// TwinCAT 3 PLC project ph_lv0
// Title: tclib_ph_lv0
// Company: Poh
// Author: Poh
// ProjectVersion: 0.1.2.0
// ProgramVersion: 3.1.4020.1
// project tree:
//   Lv0_Components/Class/ C_STREAM.TcPOU, E_SEEK_STYLE.TcDUT
//   Lv0_Components/Data Definitions/Generic Return Code/ RETURN_CODE.TcDUT, LV0_RETURNCODE.TcGVL
//   Lv0_Components/Modules/ M_TRIGGERS.TcPOU
//   Version/ Global_Version.TcGVL
// real-time tasks:
//   TASK PlcTask: cycle T#10ms, priority 20, ADS port 350
//   TASK Fast: cycle T#3ms, priority 1, ADS port 351

// ---- Lv0_Components/Class/E_SEEK_STYLE.TcDUT
{attribute 'qualified_only'}
{attribute 'strict'}
TYPE E_SEEK_STYLE :
(
	E_STREAM_BEGIN := 0,
	E_STREAM_CURRENT,
	E_STREAM_END
);
END_TYPE

// ---- Lv0_Components/Data Definitions/Generic Return Code/RETURN_CODE.TcDUT
TYPE RETURN_CODE : DINT; END_TYPE

// ---- Lv0_Components/Data Definitions/Generic Return Code/LV0_RETURNCODE.TcGVL
(*
	Y:2016	M:0005	D:0011
	Library conventions:
	Values less than 0 represent success/success code 
	Values equal to 0 represent a busy return code
	Values more than 0 represent error/error codes 
*)
{attribute 'qualified_only'}
VAR_GLOBAL CONSTANT
	RETURN_SUCCESS 	: RETURN_CODE := -1;
	RETURN_BUSY		: RETURN_CODE := 0;
	RETURN_ERROR	: RETURN_CODE := 1;
END_VAR

// ---- Version/Global_Version.TcGVL
{attribute 'TcGenerated'}
// This function has been automatically generated from the project information.
VAR_GLOBAL CONSTANT
	{attribute 'const_non_replaced'}
	{attribute 'linkalways'}
	stLibVersion_tclib_ph_lv0 : ST_LibVersion := (iMajor := 0, iMinor := 1, iBuild := 2, iRevision := 0, sVersion := '0.1.2.0');
END_VAR

// ---- Lv0_Components/Class/C_STREAM.TcPOU
FUNCTION_BLOCK C_STREAM
VAR_INPUT
END_VAR
VAR_OUTPUT
END_VAR
VAR
	_StreamSize 			: UDINT;
	_StreamData 			: POINTER TO BYTE;
	_StreamPointingPosition	: UDINT;
END_VAR

PROPERTY Base_Data : POINTER TO BYTE
GET
Base_Data := _StreamData;
END_GET
SET
_StreamData := Base_Data;
END_SET
END_PROPERTY

METHOD Clear : RETURN_CODE
VAR_INPUT
END_VAR
VAR
	_i : UDINT;
END_VAR
FOR _i := 0 TO THIS^._StreamSize - 1 BY 1 DO
	THIS^._StreamData[_i] := 0;
END_FOR
_StreamPointingPosition := 0;
_StreamFilledPosition := 0;
Clear := LV0_RETURNCODE.RETURN_SUCCESS;
END_METHOD

METHOD FB_init : BOOL
VAR_INPUT
	bInitRetains : BOOL; // if TRUE, the retain variables are initialized (warm start / cold start)
	bInCopyCode : BOOL;  // if TRUE, the instance afterwards gets moved into the copy code (online change)
	Base_Stream : POINTER TO BYTE;
	Base_StreamSize : UDINT;
END_VAR
THIS^._StreamData := Base_Stream;
THIS^._StreamSize := Base_StreamSize;
END_METHOD

METHOD Peek : Byte
VAR_INPUT
END_VAR
Peek := _StreamData[_StreamPointingPosition];
END_METHOD

PROPERTY Position : UDINT
GET
Position := _StreamPointingPosition;
END_GET
END_PROPERTY

METHOD Read : RETURN_CODE
VAR_INPUT
	OUT_DATA : POINTER TO BYTE;
	OUT_SIZE : UDINT;
END_VAR
VAR 
	_i : UDINT;
END_VAR
IF _StreamPointingPosition + OUT_SIZE > _StreamSize - 1 THEN
	Read := LV0_RETURNCODE.RETURN_ERROR;
	RETURN;
END_IF

FOR _i := 0 TO OUT_SIZE - 1 BY 1 DO
	OUT_DATA[_i] := _StreamData[_StreamPointingPosition];
	_StreamPointingPosition := _StreamPointingPosition + 1;
END_FOR
END_METHOD

METHOD Seek : RETURN_CODE
VAR_INPUT
	Offset 		: UDINT;
	SeekMode 	: E_SEEK_STYLE;
END_VAR
CASE SeekMode OF
E_SEEK_STYLE.E_STREAM_BEGIN:
	IF Offset > _StreamSize - 1 THEN
		Seek := 1 * LV0_RETURNCODE.RETURN_ERROR;
		RETURN;
	END_IF
	_StreamPointingPosition := Offset;
E_SEEK_STYLE.E_STREAM_CURRENT:
	IF _StreamPointingPosition + Offset > _StreamSize - 1 THEN
		Seek := 2 * LV0_RETURNCODE.RETURN_ERROR;
		RETURN;
	END_IF
	_StreamPointingPosition := _StreamPointingPosition + Offset;
E_SEEK_STYLE.E_STREAM_END:
	IF Offset > _StreamSize - 1 THEN
		Seek := 3 * LV0_RETURNCODE.RETURN_ERROR;
		RETURN;
	END_IF
	_StreamPointingPosition := _StreamSize - 1 - Offset;
END_CASE

Seek := LV0_RETURNCODE.RETURN_SUCCESS;
RETURN;
END_METHOD

PROPERTY Stream_Size : UDINT
GET
Stream_Size := _StreamSize;
END_GET
SET
_StreamSize := Stream_Size;
END_SET
END_PROPERTY

METHOD Write : RETURN_CODE
VAR_INPUT
	IN_DATA : POINTER TO BYTE;
	IN_SIZE : UDINT;
END_VAR
VAR 
	_i : UDINT;
END_VAR
IF _StreamPointingPosition + IN_SIZE > _StreamSize - 1 THEN
	//Buffer size insufficient.
		Write := LV0_RETURNCODE.RETURN_ERROR;
		RETURN;
END_IF

FOR _i := 0 TO IN_SIZE - 1 BY 1 DO
	_StreamData[_StreamPointingPosition] := IN_DATA[_i];
	_StreamPointingPosition := _StreamPointingPosition + 1;
END_FOR

Write := LV0_RETURNCODE.RETURN_SUCCESS;
RETURN;
END_METHOD

END_FUNCTION_BLOCK

// ---- Lv0_Components/Modules/M_TRIGGERS.TcPOU
(*
	Y:2016		M:05		D:20
	T:MODULE	N:TRIGGERS
	D:Coverts a boolean signal into R/F edge signals
*)
FUNCTION_BLOCK M_TRIGGERS
VAR_INPUT
	//SIGNAL INPUT
		BOOL_IN : BOOL;
END_VAR
VAR_OUTPUT
	//SIGNAL RISING EDGE TRIGGER
		BOOL_R : BOOL;
	//SIGNAL FALLING EDGE TRIGGER
		BOOL_F : BOOL;
	//SIGNAL RISING OR FALLING EDGE TRIGGER
		BOOL_RF: BOOL;
END_VAR
VAR
	//INTERNAL 
		_latch : BOOL;
		//UNUSED
			//SYSTEM STANDARD FUNCTION BLOCKS
			//	fb_TrigR : R_TRIG;
			//	fb_TrigF : F_TRIG;
END_VAR

IF _latch <> BOOL_IN THEN
	IF NOT _latch THEN
		BOOL_R	:= TRUE;
		BOOL_RF := TRUE;
	ELSE
		BOOL_F 	:= TRUE;
		BOOL_RF := TRUE;
	END_IF
ELSE
	BOOL_R 	:= FALSE;
	BOOL_F 	:= FALSE;
	BOOL_RF := FALSE;
END_IF
_latch := BOOL_IN;
//Unused
	////EDGE DETECTION
	//	fb_TrigR(CLK:= BOOL_IN);
	//	fb_TrigF(CLK:= BOOL_IN);
	////ASSIGNMENT
	//	BOOL_R := fb_TrigR.Q;
	//	BOOL_F := fb_TrigF.Q;
	//	BOOL_RF := fb_TrigR.Q OR fb_TrigF.Q;

END_FUNCTION_BLOCK
